(* PLC project  *)

PROGRAM MySfcProgram

END_PROGRAM
